(* Logix 5000 project; controller Tanque Emulate 5570 rev 16.30; software revision 16.03 *)

TASK MainTask (continuous, watchdog 500 ms) : MainProgram

MODULES
   Local : Emulate 5570 (ICP 3, rev 16.30)
END_MODULES

PROGRAM MainProgram   (* main routine MainRoutine *)
VAR
   B1 : BOOL;
   B2 : BOOL;
   EV : BOOL := 1;
   LLENADO : BOOL := 1;
   NIVEL : DINT := 70;
   O : BOOL;
   POWER : BOOL;
   TIMER : TIMER := (PRE := 1000);
   VACIADO : BOOL;
END_VAR

ROUTINE MainRoutine   (* ladder *)
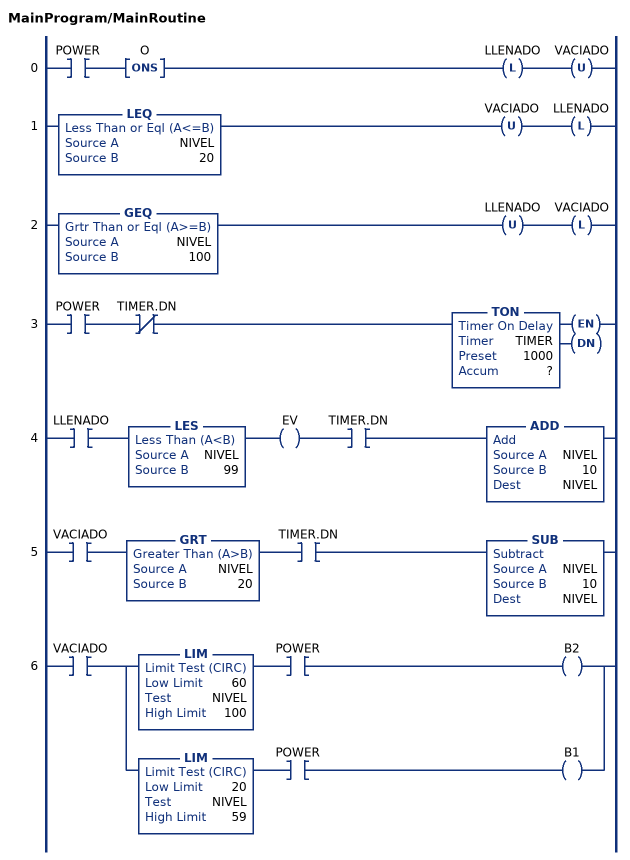
   0: XIC(POWER)ONS(O)OTL(LLENADO)OTU(VACIADO);
   1: LEQ(NIVEL,20)OTU(VACIADO)OTL(LLENADO);
   2: GEQ(NIVEL,100)OTU(LLENADO)OTL(VACIADO);
   3: XIC(POWER)XIO(TIMER.DN)TON(TIMER,?,?);
   4: XIC(LLENADO)LES(NIVEL,99)OTE(EV)XIC(TIMER.DN)ADD(NIVEL,10,NIVEL);
   5: XIC(VACIADO)GRT(NIVEL,20)XIC(TIMER.DN)SUB(NIVEL,10,NIVEL);
   6: XIC(VACIADO)[LIM(60,NIVEL,100) XIC(POWER) OTE(B2) ,LIM(20,NIVEL,59) XIC(POWER) OTE(B1) ];
END_ROUTINE
END_PROGRAM
